// TIA Portal V20 export
DATA_BLOCK "HMI_Interface_Overview"   // DB276
// stored: Access Published, MemoryReserve 100
   VAR
      State : Struct
         "Anode Reel Cut" : "HMI_IF_OverView_Unit_UDT";
         "Cathode Reel Cut" : "HMI_IF_OverView_Unit_UDT";
         "Stacker #1" : "HMI_IF_OverView_Unit_UDT";
         "Stacker #2" : "HMI_IF_OverView_Unit_UDT";
         Inspection : "HMI_IF_OverView_Unit_UDT";
      END_STRUCT;
   END_VAR
BEGIN
END_DATA_BLOCK
